TYPE ST_ExtractiveControlValveCommands :
STRUCT
	openPercentage : DINT;
	calibrate : BOOL;
	stopCalibration : BOOL;
	requireCalibration : BOOL;
END_STRUCT
END_TYPE

(* stored: Version 1.1.0.1, ProductVersion 3.1.4024.9
   DUT ST_ExtractiveControlValveCommands: Id {03f6f0f3-9c41-46ba-ad4a-a65744171dba} *)
